{attribute 'linkalways'} 
{attribute 'no_explicit_call' := 'This FB is a CLASS and must be accessed using methods or properties'}
{attribute 'enable_dynamic_creation'}
FUNCTION_BLOCK ABSTRACT AliasDatatypeBase EXTENDS UserDefinedDatatypeBase IMPLEMENTS I_AliasDatatype
VAR
	_baseDatatype : I_Datatype; // this value is the single level down
	_rootDatatype : I_Datatype; // this value is the very root of the alias (i.e. if there are stacked alias)
END_VAR

METHOD PROTECTED AddBaseDatatype
VAR_INPUT
	BaseType : I_Datatype;
END_VAR
VAR
	current : I_AliasDatatype;
	root : I_AliasDatatype;
END_VAR
IF BaseType = 0 THEN
	RETURN;
END_IF

_baseDatatype := BaseType;

// find root datatype
current := THIS^;
WHILE (TRUE) DO
	IF current.BaseDatatype.TryResolveAsAliasDatatype(root) THEN
		current := root;
		CONTINUE;
	END_IF
	EXIT;
END_WHILE
_rootDatatype := current.BaseDatatype;
END_METHOD

PROPERTY PUBLIC BaseDatatype : I_Datatype
GET
BaseDatatype := _baseDatatype;
END_GET
END_PROPERTY

METHOD PUBLIC IsEquivalentTo : BOOL
VAR_INPUT
	Datatype : I_Datatype;
END_VAR
IsEquivalentTo := Root.IsEquivalentTo(Datatype.Root);
END_METHOD

METHOD PROTECTED OnSerializeTypeWith
VAR_INPUT
	Serializer : I_Serializer;
END_VAR
SUPER^.OnSerializeTypeWith(Serializer);
Serializer.AddKey('baseDatatype');
_baseDatatype.SerializeTypeWith(Serializer);
END_METHOD

PROPERTY PUBLIC Root : I_Datatype
GET
Root := _rootDatatype;
END_GET
END_PROPERTY

METHOD PUBLIC SerializeWith
VAR_INPUT
	Serializer : I_Serializer;
END_VAR
_baseDatatype.SerializeWith(Serializer);
END_METHOD

METHOD PUBLIC TryConvertTo : BOOL
VAR_INPUT
	Destination : ANY;
END_VAR
TryConvertTo := _baseDatatype.TryConvertTo(Destination);
END_METHOD

METHOD PUBLIC TryConvertTo_ : BOOL
VAR_INPUT
	Destination : I_Datatype;
END_VAR
TryConvertTo_ := _baseDatatype.TryConvertTo_(Destination);
END_METHOD

METHOD TryDeserializeFrom : BOOL
VAR_INPUT
	Deserializer : I_Deserializer;
	Feedback : I_DeserializerFeedback;
END_VAR
TryDeserializeFrom := _baseDatatype.TryDeserializeFrom(Deserializer, Feedback);
END_METHOD

METHOD PUBLIC TryResolveAsAliasDatatype : BOOL
VAR_INPUT
	Destination : REFERENCE TO I_AliasDatatype;
END_VAR
Destination := THIS^;
TryResolveAsAliasDatatype := TRUE;
END_METHOD

PROPERTY PUBLIC TypeName : T_MAXSTRING
GET
TypeName := 'ALIAS';
END_GET
END_PROPERTY

END_FUNCTION_BLOCK

(* stored: Version 1.1.0.1, ProductVersion 3.1.4024.15
   POU AliasDatatypeBase: Id {43071a06-31c8-0f0a-109c-de25a9d3f60c}, SpecialFunc None
   Folder Protected: Id {8bcbadc5-1286-0925-29fb-ad6c7c42c3d1}
   Method AddBaseDatatype: Id {18d20a6b-4543-052d-33d0-7c44d75f8c6a}
   Property BaseDatatype: Id {34002056-d771-048e-2dbb-e738f41b9379}
   Get Get: Id {83058773-13f2-0922-3fa7-3fcabadd970a}
   Method IsEquivalentTo: Id {b65879f0-85bf-0aec-098c-0d662c3422ba}
   Method OnSerializeTypeWith: Id {50c21e86-9c66-0865-337d-e5624a0cbf3e}
   Property Root: Id {5daf7fde-382b-091c-2b1a-0472083e4613}
   Get Get: Id {e8905f4d-2aa1-0f12-0600-df6a7ba7d064}
   Method SerializeWith: Id {6182b564-094c-0830-0faf-6a2ab85fdfd7}
   Method TryConvertTo: Id {02422975-ccef-0c83-042d-6f1bb93680f4}
   Method TryConvertTo_: Id {289afa96-33fe-02e7-1e69-c25fdb7d7a42}
   Method TryDeserializeFrom: Id {83d0bd14-f34c-082f-0c86-6c1c312393f9}
   Method TryResolveAsAliasDatatype: Id {d01f897f-af3a-03be-1fac-fb410ae8769f}
   Property TypeName: Id {f78c7312-2770-0d3c-1301-f0483081b397}
   Get Get: Id {cf514327-118a-0a54-310a-8f24b17b6036} *)
